// LS Electric XG5000 project: test1112
// PLC NewPLC
// module base 0 slot 0: 입출력 모듈:XBC-DR14E (DC 24V 입력 8점, 릴레이 출력 6점)

PROGRAM NewProgram (task: 스캔 프로그램)

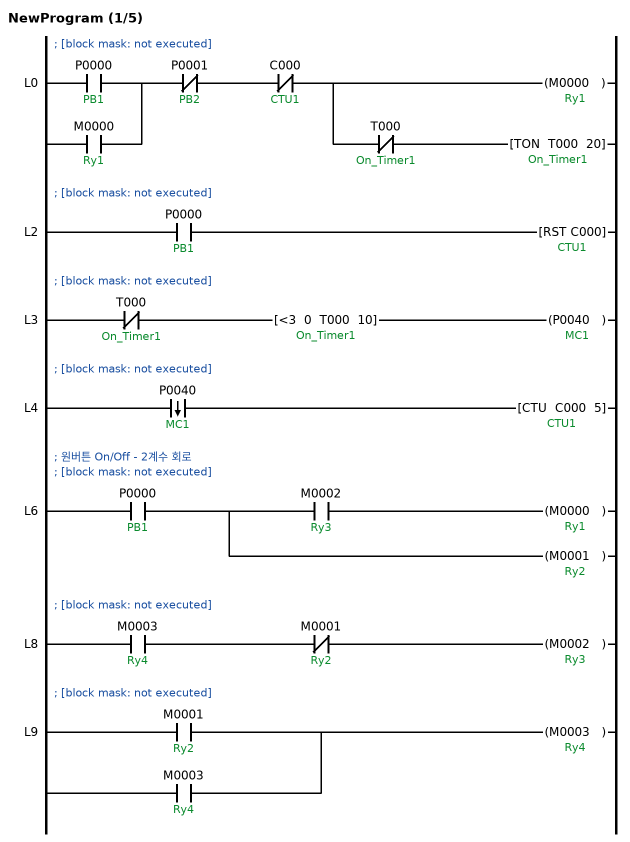
; L0 (block mask: not executed)
LOAD      P0000	// PB1
OR        M0000	// Ry1
AND NOT   P0001	// PB2
AND NOT   C000	// CTU1
OUT       M0000	// Ry1
AND NOT   T000	// On_Timer1
TON       T000 20	// On_Timer1
; L2 (block mask: not executed)
LOAD      P0000	// PB1
RST       C000	// CTU1
; L3 (block mask: not executed)
LOAD NOT  T000	// On_Timer1
AND<3     0 T000 10	// On_Timer1
OUT       P0040	// MC1
; L4 (block mask: not executed)
LOADN     P0040	// MC1
CTU       C000 5	// CTU1
// 원버튼 On/Off - 2계수 회로
; L6 (block mask: not executed)
LOAD      P0000	// PB1
MPUSH
AND       M0002	// Ry3
OUT       M0000	// Ry1
MPOP
OUT       M0001	// Ry2
; L8 (block mask: not executed)
LOAD      M0003	// Ry4
AND NOT   M0001	// Ry2
OUT       M0002	// Ry3
; L9 (block mask: not executed)
LOAD      M0001	// Ry2
OR        M0003	// Ry4
OUT       M0003	// Ry4

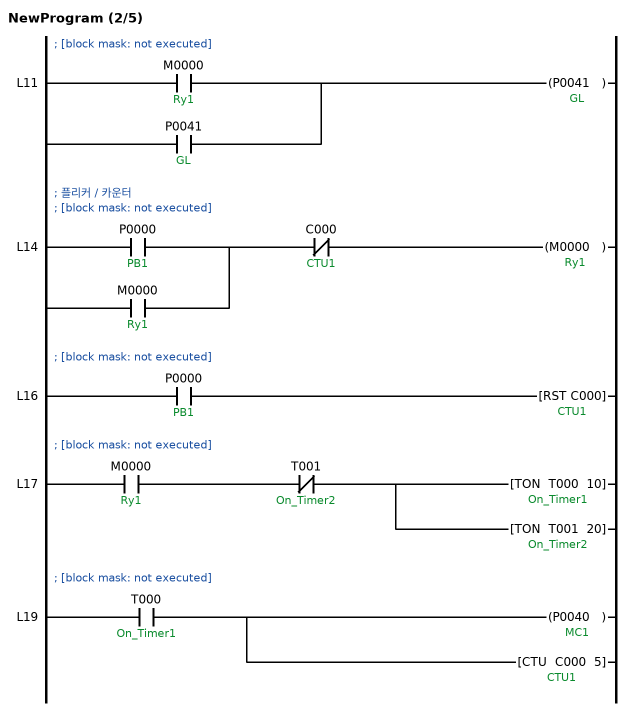
; L11 (block mask: not executed)
LOAD      M0000	// Ry1
OR        P0041	// GL
OUT       P0041	// GL
// 플리커 / 카운터
; L14 (block mask: not executed)
LOAD      P0000	// PB1
OR        M0000	// Ry1
AND NOT   C000	// CTU1
OUT       M0000	// Ry1
; L16 (block mask: not executed)
LOAD      P0000	// PB1
RST       C000	// CTU1
; L17 (block mask: not executed)
LOAD      M0000	// Ry1
AND NOT   T001	// On_Timer2
TON       T000 10	// On_Timer1
TON       T001 20	// On_Timer2
; L19 (block mask: not executed)
LOAD      T000	// On_Timer1
OUT       P0040	// MC1
CTU       C000 5	// CTU1

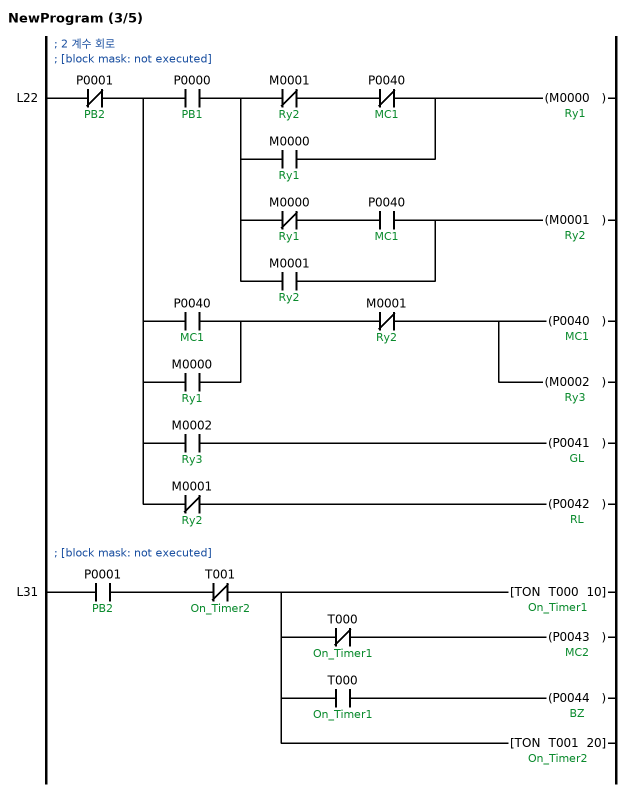
// 2 계수 회로 
; L22 (block mask: not executed)
LOAD NOT  P0001	// PB2
MPUSH
AND       P0000	// PB1
MPUSH
LOAD NOT  M0001	// Ry2
AND NOT   P0040	// MC1
OR        M0000	// Ry1
AND LOAD
OUT       M0000	// Ry1
MPOP
LOAD NOT  M0000	// Ry1
AND       P0040	// MC1
OR        M0001	// Ry2
AND LOAD
OUT       M0001	// Ry2
MLOAD
LOAD      P0040	// MC1
OR        M0000	// Ry1
AND LOAD
AND NOT   M0001	// Ry2
OUT       P0040	// MC1
OUT       M0002	// Ry3
MLOAD
AND       M0002	// Ry3
OUT       P0041	// GL
MPOP
AND NOT   M0001	// Ry2
OUT       P0042	// RL
; L31 (block mask: not executed)
LOAD      P0001	// PB2
AND NOT   T001	// On_Timer2
TON       T000 10	// On_Timer1
MPUSH
AND NOT   T000	// On_Timer1
OUT       P0043	// MC2
MLOAD
AND       T000	// On_Timer1
OUT       P0044	// BZ
MPOP
TON       T001 20	// On_Timer2

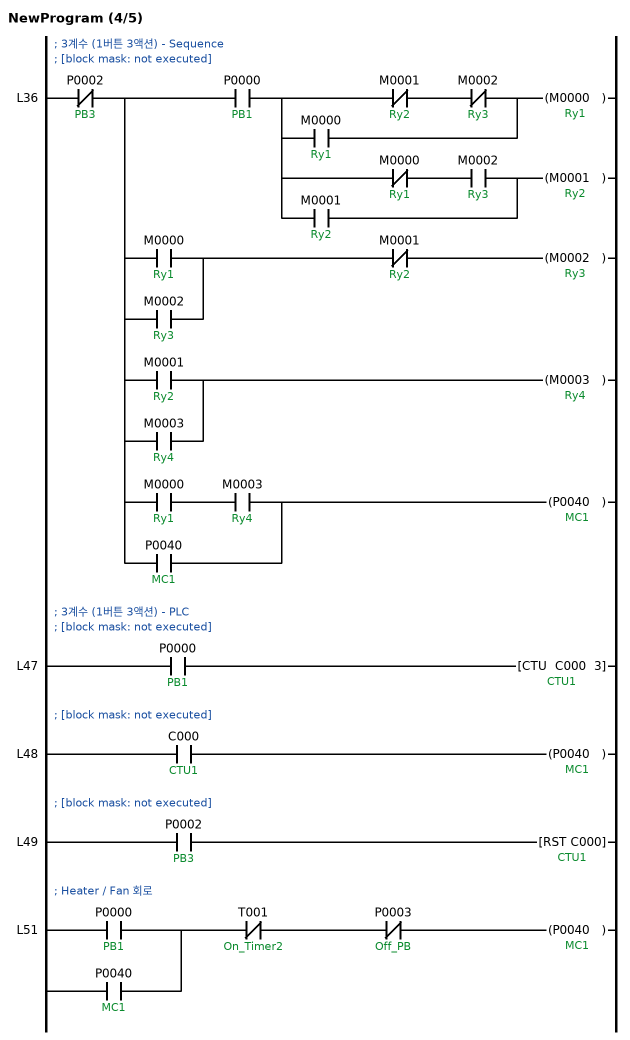
// 3계수 (1버튼 3액션) - Sequence
; L36 (block mask: not executed)
LOAD NOT  P0002	// PB3
MPUSH
AND       P0000	// PB1
MPUSH
LOAD NOT  M0001	// Ry2
AND NOT   M0002	// Ry3
OR        M0000	// Ry1
AND LOAD
OUT       M0000	// Ry1
MPOP
LOAD NOT  M0000	// Ry1
AND       M0002	// Ry3
OR        M0001	// Ry2
AND LOAD
OUT       M0001	// Ry2
MLOAD
LOAD      M0000	// Ry1
OR        M0002	// Ry3
AND LOAD
AND NOT   M0001	// Ry2
OUT       M0002	// Ry3
MLOAD
LOAD      M0001	// Ry2
OR        M0003	// Ry4
AND LOAD
OUT       M0003	// Ry4
MPOP
LOAD      M0000	// Ry1
AND       M0003	// Ry4
OR        P0040	// MC1
AND LOAD
OUT       P0040	// MC1
// 3계수 (1버튼 3액션) - PLC
; L47 (block mask: not executed)
LOAD      P0000	// PB1
CTU       C000 3	// CTU1
; L48 (block mask: not executed)
LOAD      C000	// CTU1
OUT       P0040	// MC1
; L49 (block mask: not executed)
LOAD      P0002	// PB3
RST       C000	// CTU1
// Heater / Fan 회로
; L51
LOAD      P0000	// PB1
OR        P0040	// MC1
AND NOT   T001	// On_Timer2
AND NOT   P0003	// Off_PB
OUT       P0040	// MC1

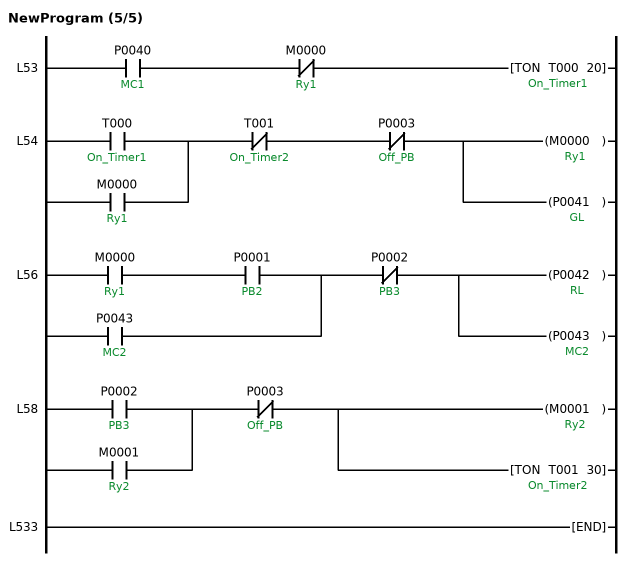
; L53
LOAD      P0040	// MC1
AND NOT   M0000	// Ry1
TON       T000 20	// On_Timer1
; L54
LOAD      T000	// On_Timer1
OR        M0000	// Ry1
AND NOT   T001	// On_Timer2
AND NOT   P0003	// Off_PB
OUT       M0000	// Ry1
OUT       P0041	// GL
; L56
LOAD      M0000	// Ry1
AND       P0001	// PB2
OR        P0043	// MC2
AND NOT   P0002	// PB3
OUT       P0042	// RL
OUT       P0043	// MC2
; L58
LOAD      P0002	// PB3
OR        M0001	// Ry2
AND NOT   P0003	// Off_PB
OUT       M0001	// Ry2
TON       T001 30	// On_Timer2
; L533
END